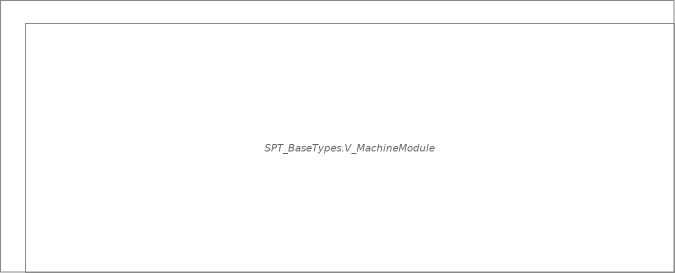
VISUALIZATION Visualization  // 675x273
    Frame (25,23 650x250)
        shows SPT_BaseTypes.V_MachineModule(HMI := MAIN.MachineModule.PackMLBaseModule_HMI)
END_VISUALIZATION

(* stored: Version 1.1.0.1, ProductVersion 3.1.4026.18
   Visu Visualization: Id {2025fc8a-0576-4fd3-84b9-241aca51007f} *)
